(* Schneider Machine Expert - Basic project modbus, file version 1.8.0.0 *)
(* ProjectInformations: Name=New project *)

HARDWARE
  Cpu 0: TM221CE16R
  EthernetConfiguration: NetworkName=M221, IpAllocationMode=FixedAddress, IpAddress=192.168.162.202, SubnetMask=255.255.255.0
  SerialLineConfiguration: Baud=Baud19200, Parity=ParityEven, DataBits=DataBits8, StopBits=StopBits1, PhysicalMedium=PhysicalMediumRs485, TransmissionMode=TransmissionModeModbusRtu, SlaveId=1, Addressing=SlaveAddressing
  MastTask: UsePeriodScanMode=false, PeriodScan=100
  FastTask: Period=255
  CpuBehavior: StartingMode=StartAsPreviousState, AutoSaveRamOnEeprom=true, WatchdogPeriod=250

SYMBOLS  (address, symbol, comment, settings)

POU New POU
  (* SectionNumber=1 *)

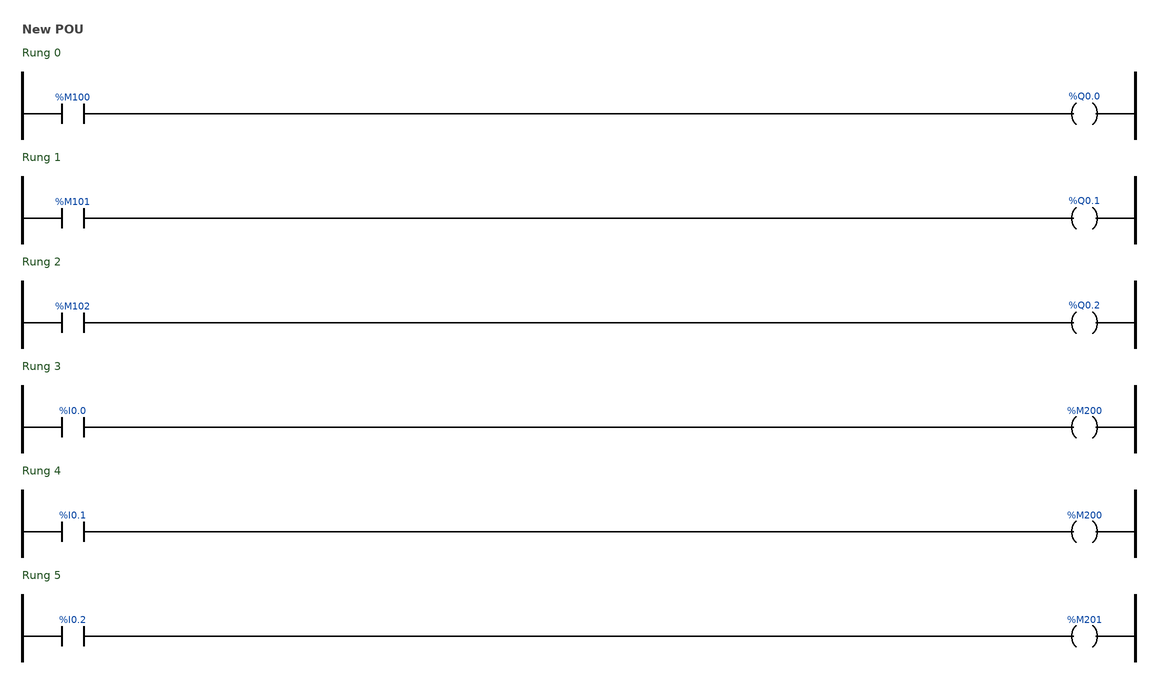

// Rung 0
  LD %M100
  ST %Q0.0
  // as ST:
  //   %Q0.0 := %M100;

// Rung 1
  LD %M101
  ST %Q0.1
  // as ST:
  //   %Q0.1 := %M101;

// Rung 2
  LD %M102
  ST %Q0.2
  // as ST:
  //   %Q0.2 := %M102;

// Rung 3
  LD %I0.0
  ST %M200
  // as ST:
  //   %M200 := %I0.0;

// Rung 4
  LD %I0.1
  ST %M200
  // as ST:
  //   %M200 := %I0.1;

// Rung 5
  LD %I0.2
  ST %M201
  // as ST:
  //   %M201 := %I0.2;
